TYPE ST_RcvDpConfig :
STRUCT
	nDpDpId			 			: UINT := 0;
	fTimeout		 			: REAL := 0.5;
	bAutoAckRei					: BOOL := TRUE;
END_STRUCT
END_TYPE

(* stored: Version 1.1.0.1, ProductVersion 3.1.4024.12
   DUT ST_RcvDpConfig: Id {203a9270-f51a-01e7-3db8-4b7478bc05b2} *)
